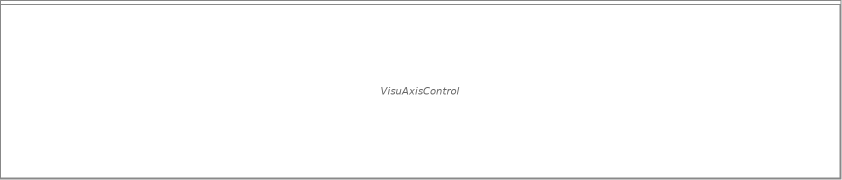
VISUALIZATION VisuAxisY  // 842x180
    Frame (0,4 840x174)
        shows VisuAxisControl(sAxisName := sAxisYName, stAxisVisu := stAxisY)
END_VISUALIZATION

(* stored: Version 1.1.0.1, ProductVersion 3.1.4022.6
   Visu VisuAxisY: Id {85a3a019-3eb0-41ea-b46b-9cd27d7d6291} *)
